FUNCTION_BLOCK INTERNAL FINAL FB_WriteRepeatedFieldMessageTests EXTENDS FB_TestSuite
VAR
    aValues : ARRAY[0..2] OF UDINT := [42, 6969, 1337];
    fbMessage : FB_TestFixed32Message;
    fbFieldCodec : FB_FieldCodecMessage(nTag:= 16#0A, ipMessage:= fbMessage);
    fbRepeatedField : FB_RepeatedField(anyArray:= F_ToAnyType(aValues), anyFirstElem:= F_ToAnyType(aValues[0]));
END_VAR

ShouldWriteNonPackedMessagesAndCalculateSize();

METHOD PRIVATE ShouldWriteNonPackedMessagesAndCalculateSize : REFERENCE TO FB_Test
VAR CONSTANT
    cExpected : ARRAY[0..20] OF BYTE := [
        16#0A, 16#05, 16#0D, 16#2A, 16#00, 16#00, 16#00,
        16#0A, 16#05, 16#0D, 16#39, 16#1B, 16#00, 16#00,
        16#0A, 16#05, 16#0D, 16#39, 16#05, 16#00, 16#00];
END_VAR
VAR_INST
    fbCtx : FB_WriteContext;
END_VAR
VAR
    aActual : ARRAY[0..20] OF BYTE;
    hr : HRESULT;
    hrSize : HRESULT;
    nSize : UDINT;
END_VAR
TEST(__POUNAME());

fbRepeatedField.InitializeFromArray(anyArray:= F_ToAnyType(aValues), anyFirstElem:= F_ToAnyType(aValues[0]), nCount:= 3);
fbCtx.FromBuffer(aActual);

hr := fbRepeatedField.WriteToWithCount(fbWriteCtx:= fbCtx, ipFieldCodec:= fbFieldCodec, nCount:= 3);
hrSize := fbRepeatedField.CalculateSize(nSize=> nSize);

AssertEquals_DINT(
    Expected:= S_OK,
    Actual:= hr,
    Message:= 'Expected repeated message write to succeed');

AssertArrayEquals_BYTE(
    Expecteds:= cExpected,
    Actuals:= aActual,
    Message:= 'Expected non-packed repeated message wire format');

AssertEquals_DINT(
    Expected:= S_OK,
    Actual:= hrSize,
    Message:= 'Expected repeated message size calculation to succeed');

AssertEquals_UDINT(
    Expected:= 21,
    Actual:= nSize,
    Message:= 'Expected non-packed repeated message size to include tags and message lengths');

TEST_FINISHED_NAMED(__POUNAME());
END_METHOD

END_FUNCTION_BLOCK

(* stored: Version 1.1.0.1
   POU FB_WriteRepeatedFieldMessageTests: Id {89bc8e78-f313-44c0-ab2f-dd749b8a02dd}, SpecialFunc None
   Method ShouldWriteNonPackedMessagesAndCalculateSize: Id {68472a16-98fd-49e5-956d-f27987d6401f} *)
